(* Logix 5000 project; controller Good_Foods_96985_10252022_1208 vendor 1 type 14 code 151 rev 32.15; software revision 32.04; part 3 of 4 *)
(* tags used below, declared in another part *)
   Active_Container_Recipe : Container_Recipe;
   AG_Index_Sys : BOOL;
   Axis_Virtual_Left_Denest : AXIS_VIRTUAL;
   Axis_Virtual_Right_Denest : AXIS_VIRTUAL;
   bAuto_Axis_Reset : BOOL;
   bAuto_Disable_Servos : BOOL;
   bAuto_Reset_Servos : BOOL;
   bHMI_IND_Servos_Disable : BOOL;
   bHMI_IND_Servos_Enable : BOOL;
   bHMI_PB_Fault_Reset : BOOL;
   bHMI_PB_JogFwd_Left_Denester : BOOL;
   bHMI_PB_JogFwd_Right_Denester : BOOL;
   bHMI_PB_JogRev_Left_Denester : BOOL;
   bHMI_PB_JogRev_Right_Denester : BOOL;
   bHMI_PB_Left_Denester_Enabled : BOOL;
   bHMI_PB_Move_Screws_to_Zero : BOOL;
   bHMI_PB_Park_Denesters : BOOL;
   bHMI_PB_Park_Left_Denester : BOOL;
   bHMI_PB_Park_Right_Denester : BOOL;
   bHMI_PB_Right_Denester_Enabled : BOOL;
   bHMI_PB_Servos_Disable : BOOL;
   bHMI_PB_Servos_Enable : BOOL;
   bHMI_PB_Teach_Zero_Left_Denester : BOOL;
   bHMI_PB_Teach_Zero_Master_Encoder : BOOL;
   bHMI_PB_Teach_Zero_Right_Denester : BOOL;
   bHMI_PB_Zero_All : BOOL;
   bHome_Master_Encoder : BOOL;
   bLeft_Index_Complete : BOOL;
   bLeft_Index_Cycle_Duration : BOOL;
   bLeft_Indexing : BOOL;
   bLeft_System_Not_Running : BOOL;
   bLeftPrimeBacklog_OK : BOOL;
   bMachine_Startup_Delay : BOOL;
   bRight_Index_Complete : BOOL;
   bRight_Index_Cycle_Duration : BOOL;
   bRight_Indexing : BOOL;
   bRight_System_Not_Running : BOOL;
   bRightPrimeBacklog_OK : BOOL;
   bSystem_Active : BOOL;
   bSystem_Alarm_Active : BOOL;
   bSystem_Decouple_CMPLT : BOOL;
   bSystem_Denester_Run_Perm : BOOL;
   bSystem_Gearing_CMPLT : BOOL;
   bSystem_Park_CMPLT : BOOL;
   bSystem_Sync_CMPLT : BOOL;
   CamP_RampDwn : CAM_PROFILE[40];
   CamP_RampUp : CAM_PROFILE[40];
   CamP_Run : CAM_PROFILE[40];
   ctuLeftStartup : COUNTER;
   ctuRightDlyStop : COUNTER;
   DI_Safety_Relay_OK : BOOL;
   dLeft_Denester_Jog_Dir : DINT;
   dRight_Denester_Jog_Dir : DINT;
   dSystem_Start_Seq_CMD : DINT;
   dSystem_Stop_Seq_CMD : DINT;
   dTempRevsTime : DINT;
   Index_Position : INT;
   intLug_Drop_High_Limit : INT;
   Left_Denester : AXIS_CIP_DRIVE;
   Left_Index_Cycle_Duration_Timer : TIMER;
   Left_Index_Measured_Cycle_Time : DINT;
   Left_Not_Running_Timer : TIMER;
   MAFR_Axis_Virtual : MOTION_INSTRUCTION;
   MAFR_Left_Denester : MOTION_INSTRUCTION;
   MAFR_Right_Denester : MOTION_INSTRUCTION;
   MAG_StartGear_LeftDenester : MOTION_INSTRUCTION;
   MAG_StartGear_RightDenester : MOTION_INSTRUCTION;
   MAH_Axis_Virtual : MOTION_INSTRUCTION;
   MAH_Left_Denester : MOTION_INSTRUCTION;
   MAH_Master_Encoder : MOTION_INSTRUCTION;
   MAH_Right_Denester : MOTION_INSTRUCTION;
   MAJ_Left_Denester_Jog : MOTION_INSTRUCTION;
   MAJ_Right_Denester_Jog : MOTION_INSTRUCTION;
   MAM_Home_Left_Denester : MOTION_INSTRUCTION;
   MAM_Home_Right_Denester : MOTION_INSTRUCTION;
   MAM_Left_Denester_Sync : MOTION_INSTRUCTION;
   MAM_Park_Left_Denester : MOTION_INSTRUCTION;
   MAM_Park_Right_Denester : MOTION_INSTRUCTION;
   MAM_Right_Denester_Sync : MOTION_INSTRUCTION;
   mamAxisLeftSCREW_INDEXMOVE : MOTION_INSTRUCTION;
   mamAxisRightSCREW_INDEXMOVE : MOTION_INSTRUCTION;
   MAPC_LeftDenesterToLugBelt_RampDwn : MOTION_INSTRUCTION;
   MAPC_LeftDenesterToLugBelt_RampUp : MOTION_INSTRUCTION;
   MAPC_LeftDenesterToLugBelt_Run : MOTION_INSTRUCTION;
   MAPC_RightDenesterToLugBelt_RampDwn : MOTION_INSTRUCTION;
   MAPC_RightDenesterToLugBelt_RampUp : MOTION_INSTRUCTION;
   MAPC_RightDenesterToLugBelt_Run : MOTION_INSTRUCTION;
   MAS_LeftDenester : MOTION_INSTRUCTION;
   MAS_LeftDenester_Jog : MOTION_INSTRUCTION;
   MAS_LeftDenester_Virtual : MOTION_INSTRUCTION;
   MAS_RightDenester : MOTION_INSTRUCTION;
   MAS_RightDenester_Jog : MOTION_INSTRUCTION;
   MAS_RightDenester_Virtual : MOTION_INSTRUCTION;
   MAS_TEMP_Axis_Master_Follow : MOTION_INSTRUCTION;
   MASR_Axis_Virtual : MOTION_INSTRUCTION;
   MASR_Left_Denester : MOTION_INSTRUCTION;
   MASR_Master_Encoder : MOTION_INSTRUCTION;
   MASR_Right_Denester : MOTION_INSTRUCTION;
   Master_Encoder : AXIS_CIP_DRIVE;
   MRP_Axis_Virtual_Sync_Left : MOTION_INSTRUCTION;
   MRP_Axis_Virtual_Sync_Right : MOTION_INSTRUCTION;
   MSF_Left_Denester : MOTION_INSTRUCTION;
   MSF_Right_Denester : MOTION_INSTRUCTION;
   MSO_Left_Denester : MOTION_INSTRUCTION;
   MSO_Right_Denester : MOTION_INSTRUCTION;
   ONS : DINT[16];
   r_Index_Speed : REAL;
   rHMI_Jog_Speed : REAL;
   Right_Denester : AXIS_CIP_DRIVE;
   Right_Index_Cycle_Duration_Timer : TIMER;
   Right_Index_Measured_Cycle_Time : DINT;
   Right_Not_Running_Timer : TIMER;
   rJog_Speed_Command : DINT;
   rLeft_Actual_Throughput : REAL;
   rLeft_Denester_Actual_Position : REAL;
   rLeft_Denester_Position_High : REAL;
   rLeft_Denester_Position_Low : REAL;
   rMaster_Encoder_Actual_Position : REAL;
   rRight_Actual_Throughput : REAL;
   rRight_Denester_Actual_Position : REAL;
   rRight_Denester_Position_High : DINT;
   rRight_Denester_Position_Low : REAL;
   rSystem_Throughput : REAL;
   rTEMP_Axis_Master_Follow_Actual_Position : REAL;
   rVirtual_Right_Denest_Actual_Position : REAL;
   Screw_Accel : REAL;
   Screw_Decel : REAL;
   Servos : MOTION_GROUP;
   TEMP_Axis_Master_Follow : AXIS_VIRTUAL;
   tMachine_Startup_Delay : TIMER;
   tTempRevs : TIMER;
(* MainProgram, continued *)

ROUTINE _20_Servo_Init   (* ladder *)
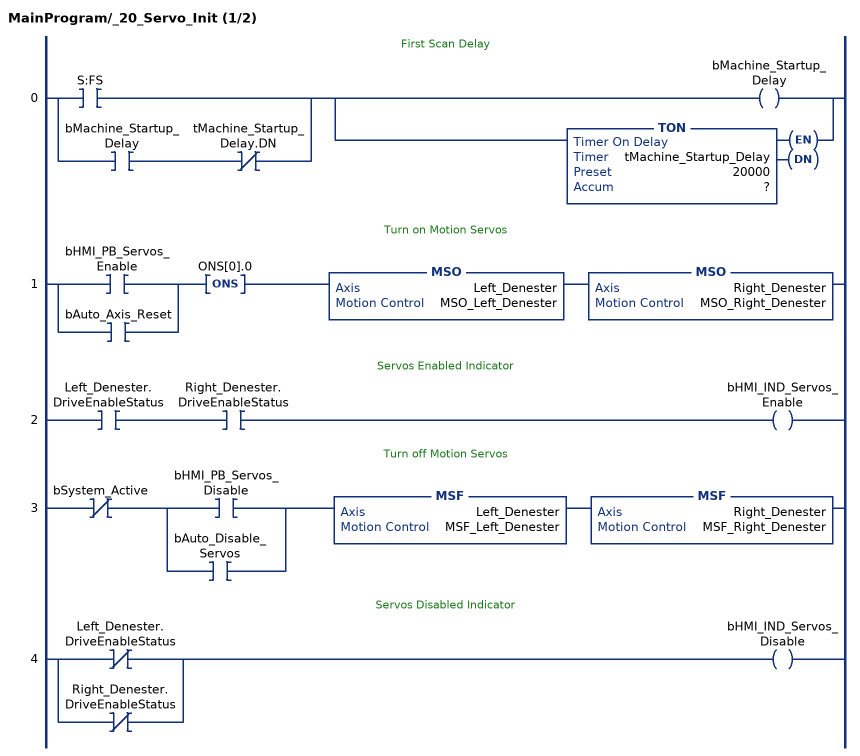
   // First Scan Delay
   0: [XIC(S:FS) ,XIC(bMachine_Startup_Delay) XIO(tMachine_Startup_Delay.DN) ][OTE(bMachine_Startup_Delay) ,TON(tMachine_Startup_Delay,?,?) ];
   // Turn on Motion Servos
   1: [XIC(bHMI_PB_Servos_Enable) ,XIC(bAuto_Axis_Reset) ]ONS(ONS[0].0)MSO(Left_Denester,MSO_Left_Denester)MSO(Right_Denester,MSO_Right_Denester);
   // Servos Enabled Indicator
   2: XIC(Left_Denester.DriveEnableStatus)XIC(Right_Denester.DriveEnableStatus)OTE(bHMI_IND_Servos_Enable);
   // Turn off Motion Servos
   3: XIO(bSystem_Active)[XIC(bHMI_PB_Servos_Disable) ,XIC(bAuto_Disable_Servos) ]MSF(Left_Denester,MSF_Left_Denester)MSF(Right_Denester,MSF_Right_Denester);
   // Servos Disabled Indicator
   4: [XIO(Left_Denester.DriveEnableStatus) ,XIO(Right_Denester.DriveEnableStatus) ]OTE(bHMI_IND_Servos_Disable);
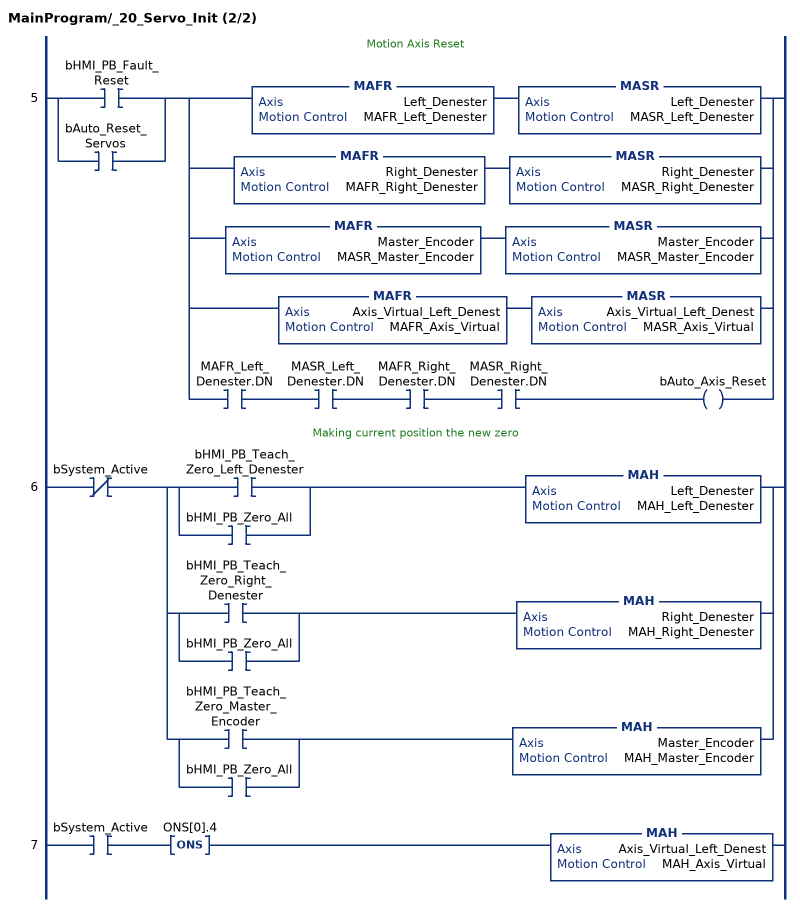
   // Motion Axis Reset
   5: [XIC(bHMI_PB_Fault_Reset) ,XIC(bAuto_Reset_Servos) ][MAFR(Left_Denester,MAFR_Left_Denester) MASR(Left_Denester,MASR_Left_Denester) ,MAFR(Right_Denester,MAFR_Right_Denester) MASR(Right_Denester,MASR_Right_Denester) ,MAFR(Master_Encoder,MASR_Master_Encoder) MASR(Master_Encoder,MASR_Master_Encoder) ,MAFR(Axis_Virtual_Left_Denest,MAFR_Axis_Virtual) MASR(Axis_Virtual_Left_Denest,MASR_Axis_Virtual) ,XIC(MAFR_Left_Denester.DN) XIC(MASR_Left_Denester.DN) XIC(MAFR_Right_Denester.DN) XIC(MASR_Right_Denester.DN) OTE(bAuto_Axis_Reset) ];
   // Making current position the new zero
   6: XIO(bSystem_Active)[[XIC(bHMI_PB_Teach_Zero_Left_Denester) ,XIC(bHMI_PB_Zero_All) ] MAH(Left_Denester,MAH_Left_Denester) ,[XIC(bHMI_PB_Teach_Zero_Right_Denester) ,XIC(bHMI_PB_Zero_All) ] MAH(Right_Denester,MAH_Right_Denester) ,[XIC(bHMI_PB_Teach_Zero_Master_Encoder) ,XIC(bHMI_PB_Zero_All) ] MAH(Master_Encoder,MAH_Master_Encoder) ];
   7: XIC(bSystem_Active)ONS(ONS[0].4)MAH(Axis_Virtual_Left_Denest,MAH_Axis_Virtual);
END_ROUTINE

ROUTINE _25_Servo_Motion   (* ladder *)
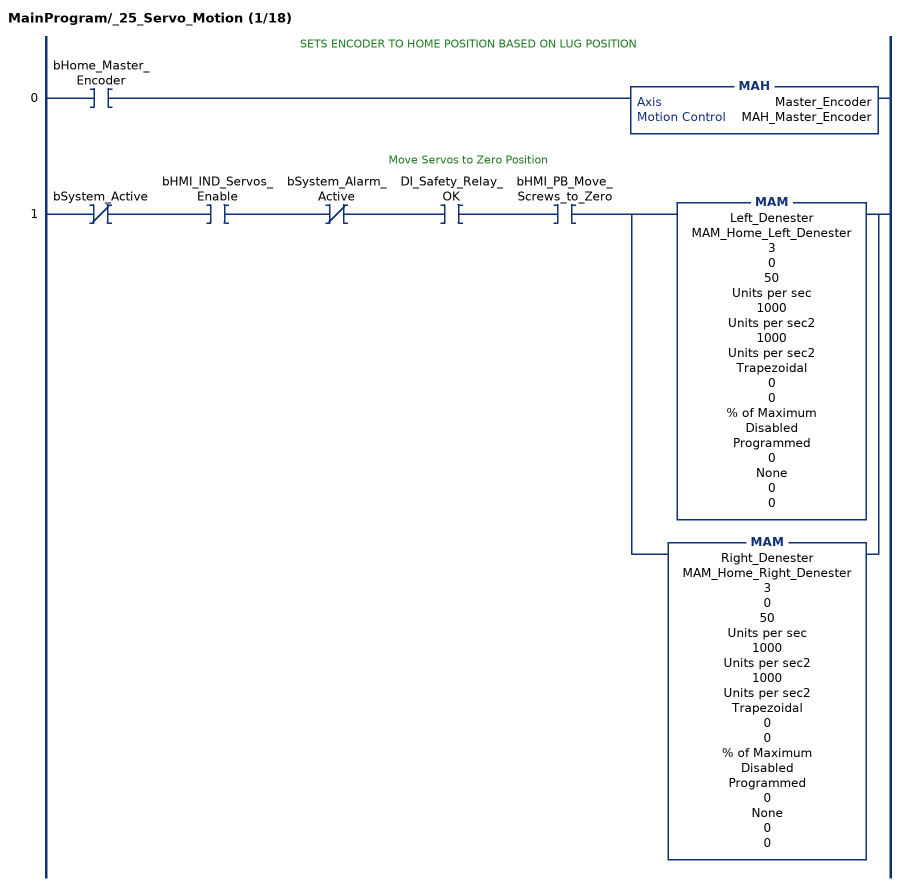
   // SETS ENCODER TO HOME POSITION BASED ON LUG POSITION
   0: XIC(bHome_Master_Encoder)MAH(Master_Encoder,MAH_Master_Encoder);
   // Move Servos to Zero Position
   1: XIO(bSystem_Active)XIC(bHMI_IND_Servos_Enable)XIO(bSystem_Alarm_Active)XIC(DI_Safety_Relay_OK)XIC(bHMI_PB_Move_Screws_to_Zero)[MAM(Left_Denester,MAM_Home_Left_Denester,3,0,50,Units per sec,1000,Units per sec2,1000,Units per sec2,Trapezoidal,0,0,% of Maximum,Disabled,Programmed,0,None,0,0) ,MAM(Right_Denester,MAM_Home_Right_Denester,3,0,50,Units per sec,1000,Units per sec2,1000,Units per sec2,Trapezoidal,0,0,% of Maximum,Disabled,Programmed,0,None,0,0) ];
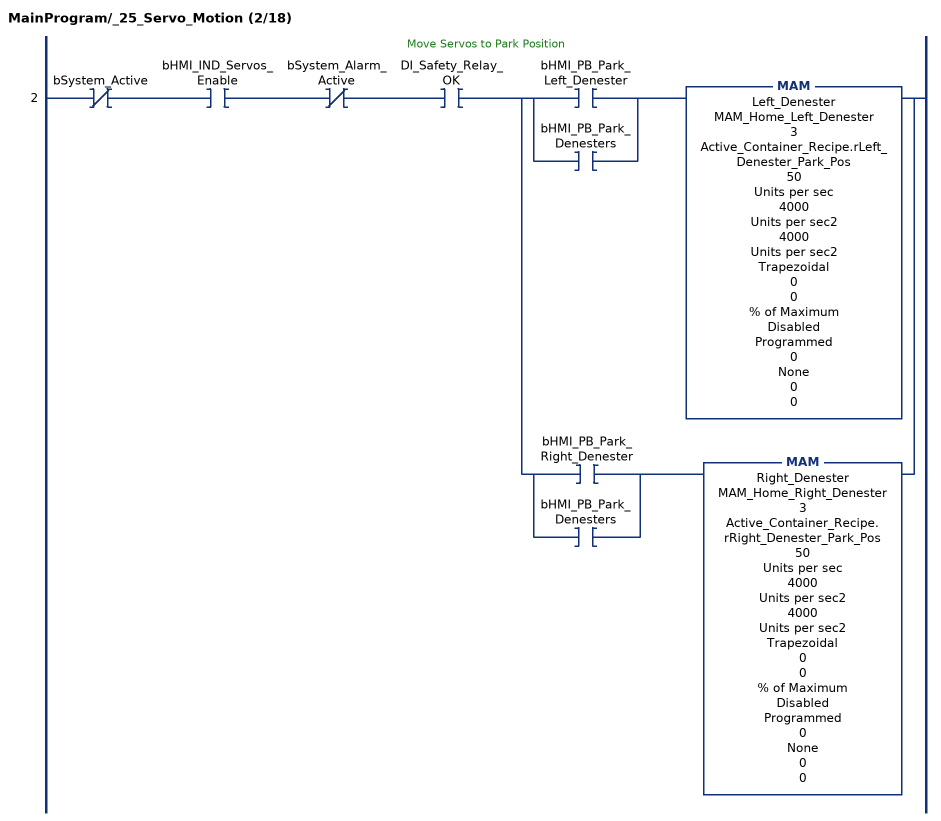
   // Move Servos to Park Position
   2: XIO(bSystem_Active)XIC(bHMI_IND_Servos_Enable)XIO(bSystem_Alarm_Active)XIC(DI_Safety_Relay_OK)[[XIC(bHMI_PB_Park_Left_Denester) ,XIC(bHMI_PB_Park_Denesters) ] MAM(Left_Denester,MAM_Home_Left_Denester,3,Active_Container_Recipe.rLeft_Denester_Park_Pos,50,Units per sec,4000,Units per sec2,4000,Units per sec2,Trapezoidal,0,0,% of Maximum,Disabled,Programmed,0,None,0,0) ,[XIC(bHMI_PB_Park_Right_Denester) ,XIC(bHMI_PB_Park_Denesters) ] MAM(Right_Denester,MAM_Home_Right_Denester,3,Active_Container_Recipe.rRight_Denester_Park_Pos,50,Units per sec,4000,Units per sec2,4000,Units per sec2,Trapezoidal,0,0,% of Maximum,Disabled,Programmed,0,None,0,0) ];
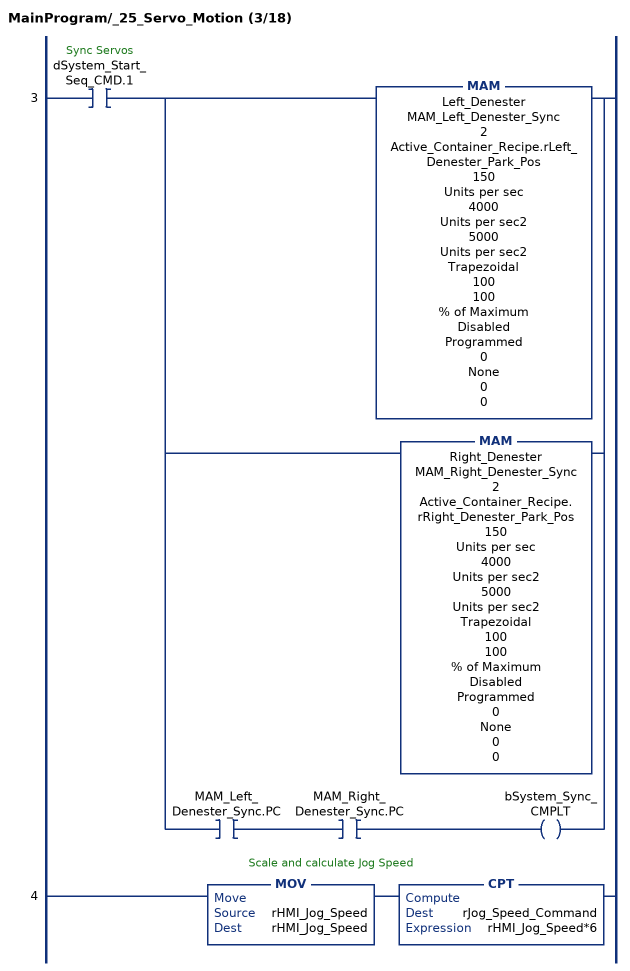
   3: XIC(dSystem_Start_Seq_CMD.1)[MAM(Left_Denester,MAM_Left_Denester_Sync,2,Active_Container_Recipe.rLeft_Denester_Park_Pos,150,Units per sec,4000,Units per sec2,5000,Units per sec2,Trapezoidal,100,100,% of Maximum,Disabled,Programmed,0,None,0,0) ,MAM(Right_Denester,MAM_Right_Denester_Sync,2,Active_Container_Recipe.rRight_Denester_Park_Pos,150,Units per sec,4000,Units per sec2,5000,Units per sec2,Trapezoidal,100,100,% of Maximum,Disabled,Programmed,0,None,0,0) ,XIC(MAM_Left_Denester_Sync.PC) XIC(MAM_Right_Denester_Sync.PC) OTE(bSystem_Sync_CMPLT) ];
   // Scale and calculate Jog Speed
   4: MOV(rHMI_Jog_Speed,rHMI_Jog_Speed)CPT(rJog_Speed_Command,rHMI_Jog_Speed*6);
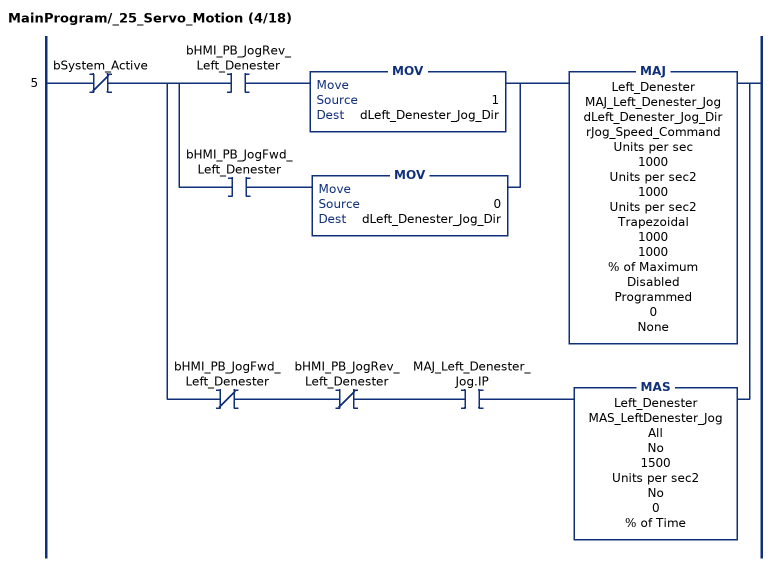
   5: XIO(bSystem_Active)[[XIC(bHMI_PB_JogRev_Left_Denester) MOV(1,dLeft_Denester_Jog_Dir) ,XIC(bHMI_PB_JogFwd_Left_Denester) MOV(0,dLeft_Denester_Jog_Dir) ] MAJ(Left_Denester,MAJ_Left_Denester_Jog,dLeft_Denester_Jog_Dir,rJog_Speed_Command,Units per sec,1000,Units per sec2,1000,Units per sec2,Trapezoidal,1000,1000,% of Maximum,Disabled,Programmed,0,None) ,XIO(bHMI_PB_JogFwd_Left_Denester) XIO(bHMI_PB_JogRev_Left_Denester) XIC(MAJ_Left_Denester_Jog.IP) MAS(Left_Denester,MAS_LeftDenester_Jog,All,No,1500,Units per sec2,No,0,% of Time) ];
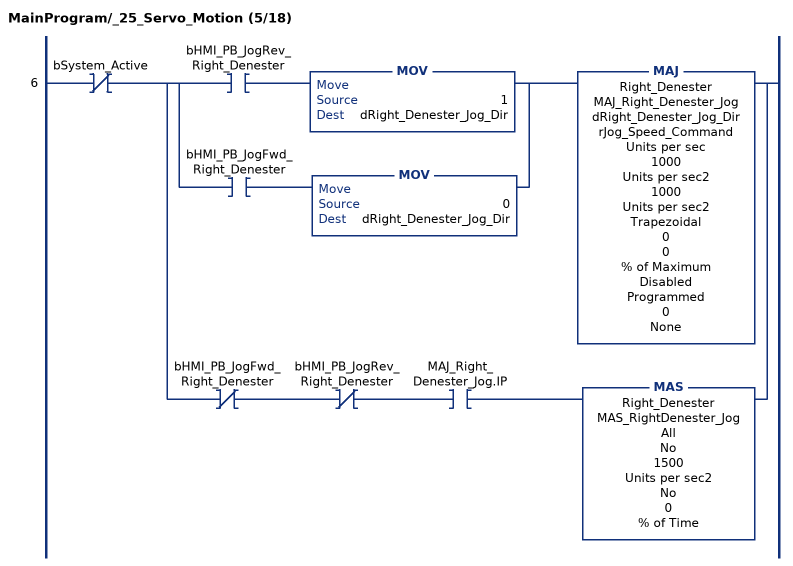
   6: XIO(bSystem_Active)[[XIC(bHMI_PB_JogRev_Right_Denester) MOV(1,dRight_Denester_Jog_Dir) ,XIC(bHMI_PB_JogFwd_Right_Denester) MOV(0,dRight_Denester_Jog_Dir) ] MAJ(Right_Denester,MAJ_Right_Denester_Jog,dRight_Denester_Jog_Dir,rJog_Speed_Command,Units per sec,1000,Units per sec2,1000,Units per sec2,Trapezoidal,0,0,% of Maximum,Disabled,Programmed,0,None) ,XIO(bHMI_PB_JogFwd_Right_Denester) XIO(bHMI_PB_JogRev_Right_Denester) XIC(MAJ_Right_Denester_Jog.IP) MAS(Right_Denester,MAS_RightDenester_Jog,All,No,1500,Units per sec2,No,0,% of Time) ];
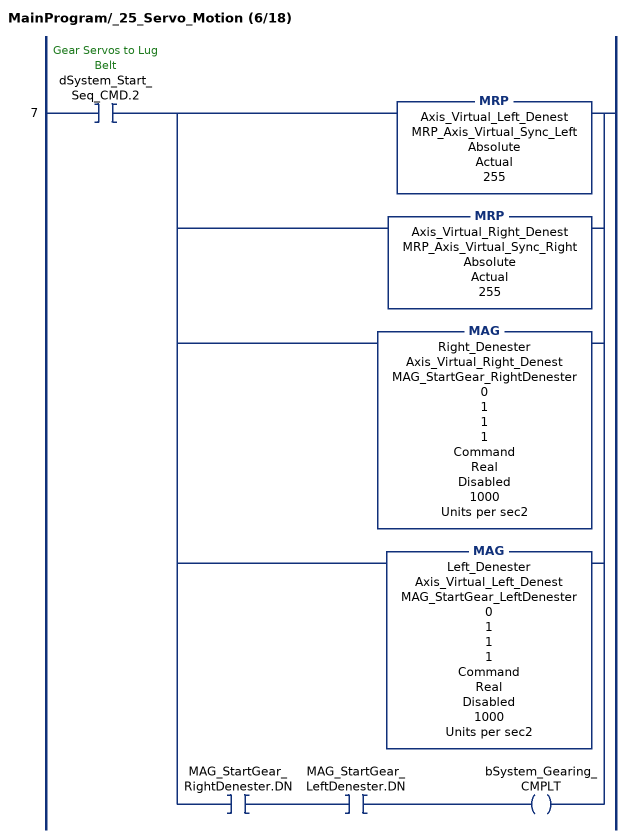
   7: XIC(dSystem_Start_Seq_CMD.2)[MRP(Axis_Virtual_Left_Denest,MRP_Axis_Virtual_Sync_Left,Absolute,Actual,255) ,MRP(Axis_Virtual_Right_Denest,MRP_Axis_Virtual_Sync_Right,Absolute,Actual,255) ,MAG(Right_Denester,Axis_Virtual_Right_Denest,MAG_StartGear_RightDenester,0,1,1,1,Command,Real,Disabled,1000,Units per sec2) ,MAG(Left_Denester,Axis_Virtual_Left_Denest,MAG_StartGear_LeftDenester,0,1,1,1,Command,Real,Disabled,1000,Units per sec2) ,XIC(MAG_StartGear_RightDenester.DN) XIC(MAG_StartGear_LeftDenester.DN) OTE(bSystem_Gearing_CMPLT) ];
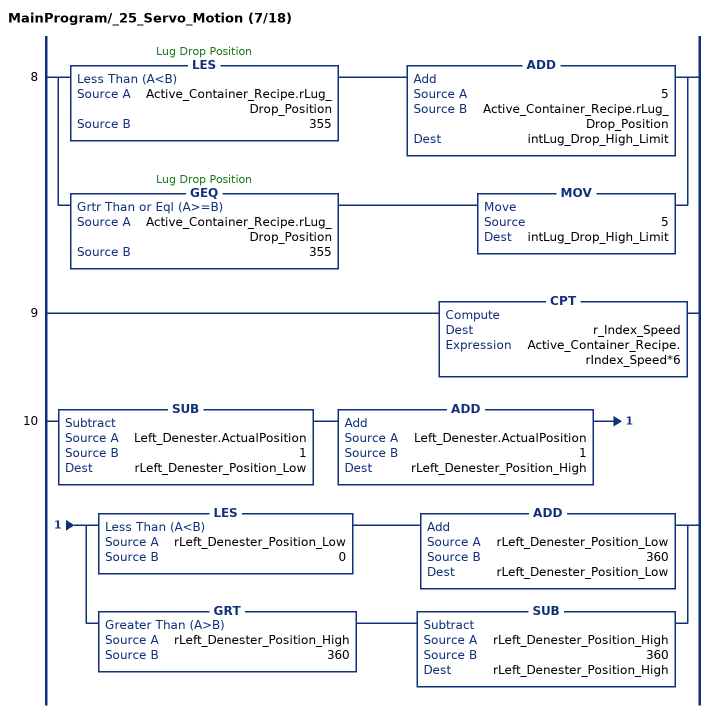
   8: [LES(Active_Container_Recipe.rLug_Drop_Position,355) ADD(5,Active_Container_Recipe.rLug_Drop_Position,intLug_Drop_High_Limit) ,GEQ(Active_Container_Recipe.rLug_Drop_Position,355) MOV(5,intLug_Drop_High_Limit) ];
   9: CPT(r_Index_Speed,Active_Container_Recipe.rIndex_Speed*6);
   10: SUB(Left_Denester.ActualPosition,1,rLeft_Denester_Position_Low)ADD(Left_Denester.ActualPosition,1,rLeft_Denester_Position_High)[LES(rLeft_Denester_Position_Low,0) ADD(rLeft_Denester_Position_Low,360,rLeft_Denester_Position_Low) ,GRT(rLeft_Denester_Position_High,360) SUB(rLeft_Denester_Position_High,360,rLeft_Denester_Position_High) ];
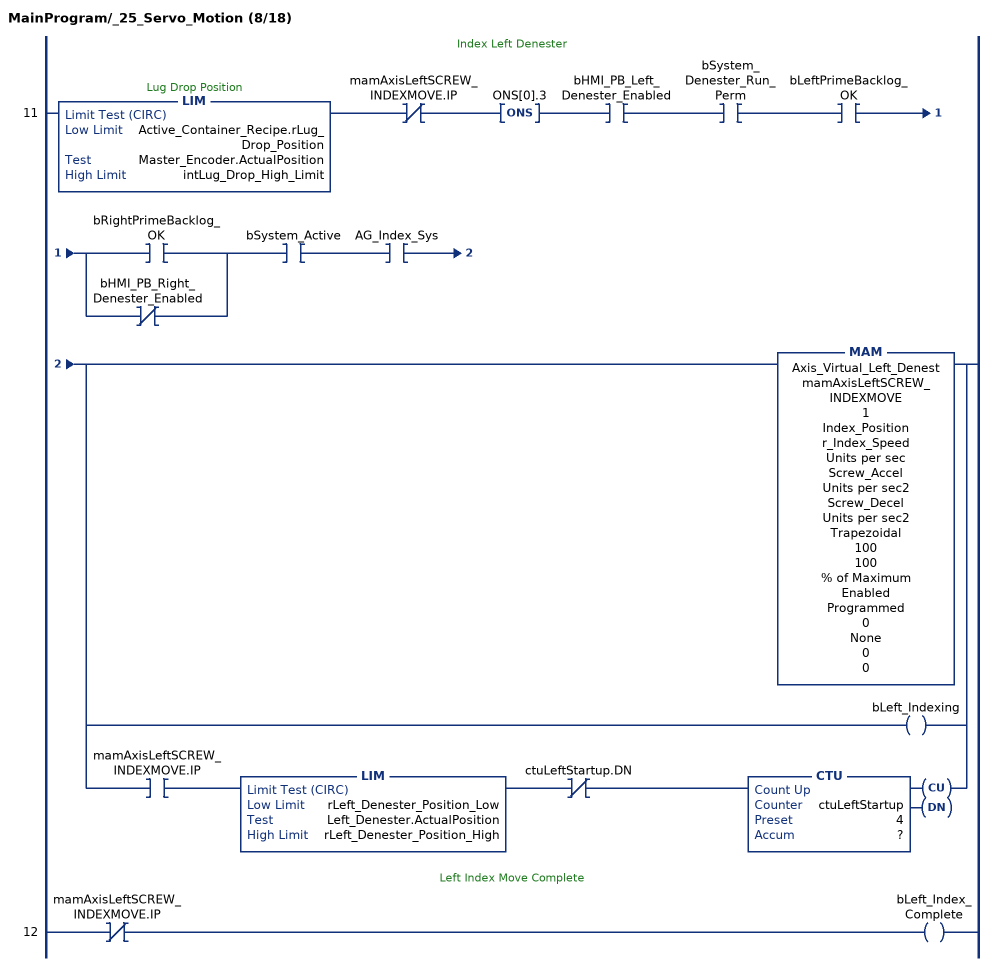
   // Index Left Denester
   11: LIM(Active_Container_Recipe.rLug_Drop_Position,Master_Encoder.ActualPosition,intLug_Drop_High_Limit)XIO(mamAxisLeftSCREW_INDEXMOVE.IP)ONS(ONS[0].3)XIC(bHMI_PB_Left_Denester_Enabled)XIC(bSystem_Denester_Run_Perm)XIC(bLeftPrimeBacklog_OK)[XIC(bRightPrimeBacklog_OK) ,XIO(bHMI_PB_Right_Denester_Enabled) ]XIC(bSystem_Active)XIC(AG_Index_Sys)[MAM(Axis_Virtual_Left_Denest,mamAxisLeftSCREW_INDEXMOVE,1,Index_Position,r_Index_Speed,Units per sec,Screw_Accel,Units per sec2,Screw_Decel,Units per sec2,Trapezoidal,100,100,% of Maximum,Enabled,Programmed,0,None,0,0) ,OTE(bLeft_Indexing) ,XIC(mamAxisLeftSCREW_INDEXMOVE.IP) LIM(rLeft_Denester_Position_Low,Left_Denester.ActualPosition,rLeft_Denester_Position_High) XIO(ctuLeftStartup.DN) CTU(ctuLeftStartup,?,?) ];
   // Left Index Move Complete
   12: XIO(mamAxisLeftSCREW_INDEXMOVE.IP)OTE(bLeft_Index_Complete);
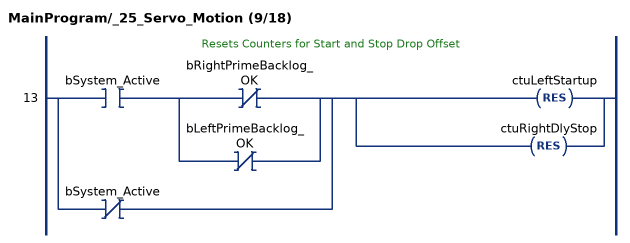
   // Resets Counters for Start and Stop Drop Offset
   13: [XIC(bSystem_Active) [XIO(bRightPrimeBacklog_OK) ,XIO(bLeftPrimeBacklog_OK) ] ,XIO(bSystem_Active) ][RES(ctuLeftStartup) ,RES(ctuRightDlyStop) ];
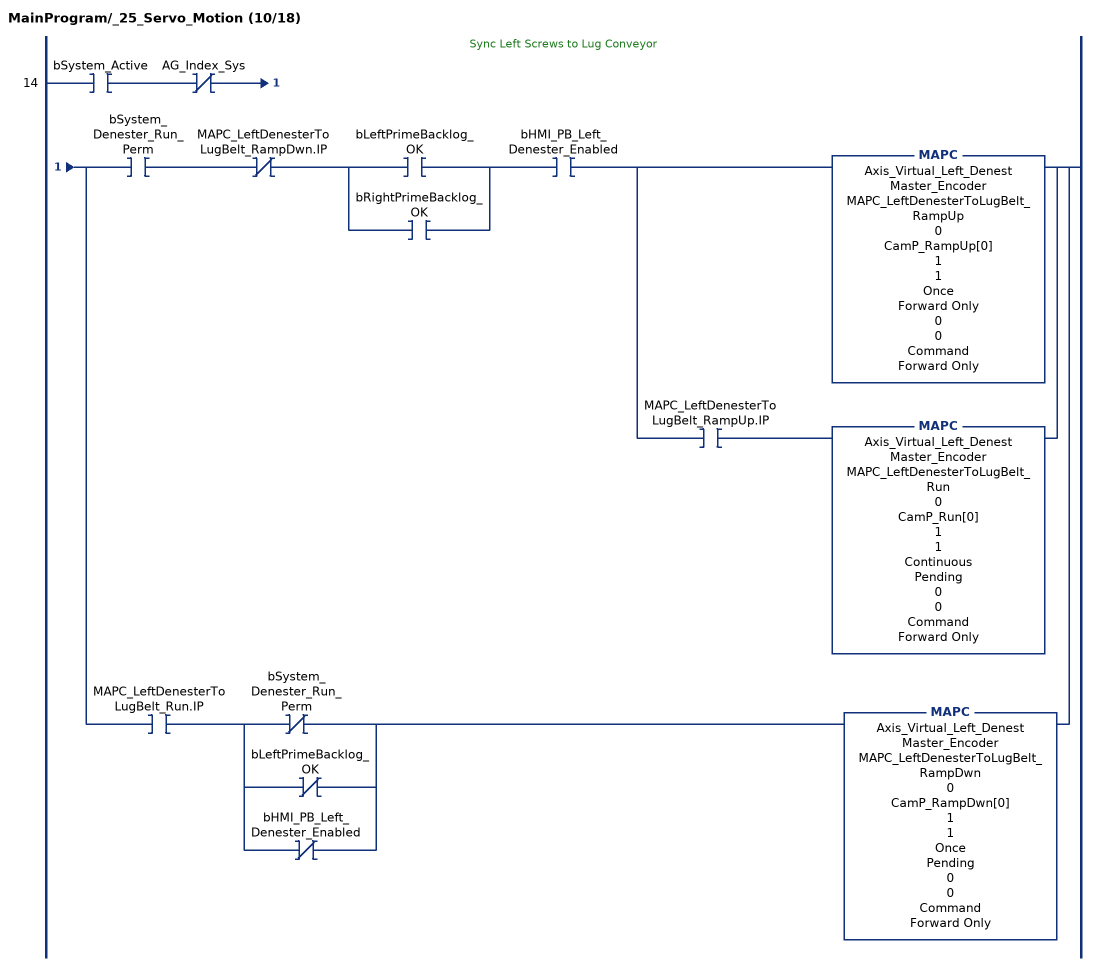
   // Sync Left Screws to Lug Conveyor
   14: XIC(bSystem_Active)XIO(AG_Index_Sys)[XIC(bSystem_Denester_Run_Perm) XIO(MAPC_LeftDenesterToLugBelt_RampDwn.IP) [XIC(bLeftPrimeBacklog_OK) ,XIC(bRightPrimeBacklog_OK) ] XIC(bHMI_PB_Left_Denester_Enabled) [MAPC(Axis_Virtual_Left_Denest,Master_Encoder,MAPC_LeftDenesterToLugBelt_RampUp,0,CamP_RampUp[0],1,1,Once,Forward Only,0,0,Command,Forward Only) ,XIC(MAPC_LeftDenesterToLugBelt_RampUp.IP) MAPC(Axis_Virtual_Left_Denest,Master_Encoder,MAPC_LeftDenesterToLugBelt_Run,0,CamP_Run[0],1,1,Continuous,Pending,0,0,Command,Forward Only) ] ,XIC(MAPC_LeftDenesterToLugBelt_Run.IP) [XIO(bSystem_Denester_Run_Perm) ,XIO(bLeftPrimeBacklog_OK) ,XIO(bHMI_PB_Left_Denester_Enabled) ] MAPC(Axis_Virtual_Left_Denest,Master_Encoder,MAPC_LeftDenesterToLugBelt_RampDwn,0,CamP_RampDwn[0],1,1,Once,Pending,0,0,Command,Forward Only) ];
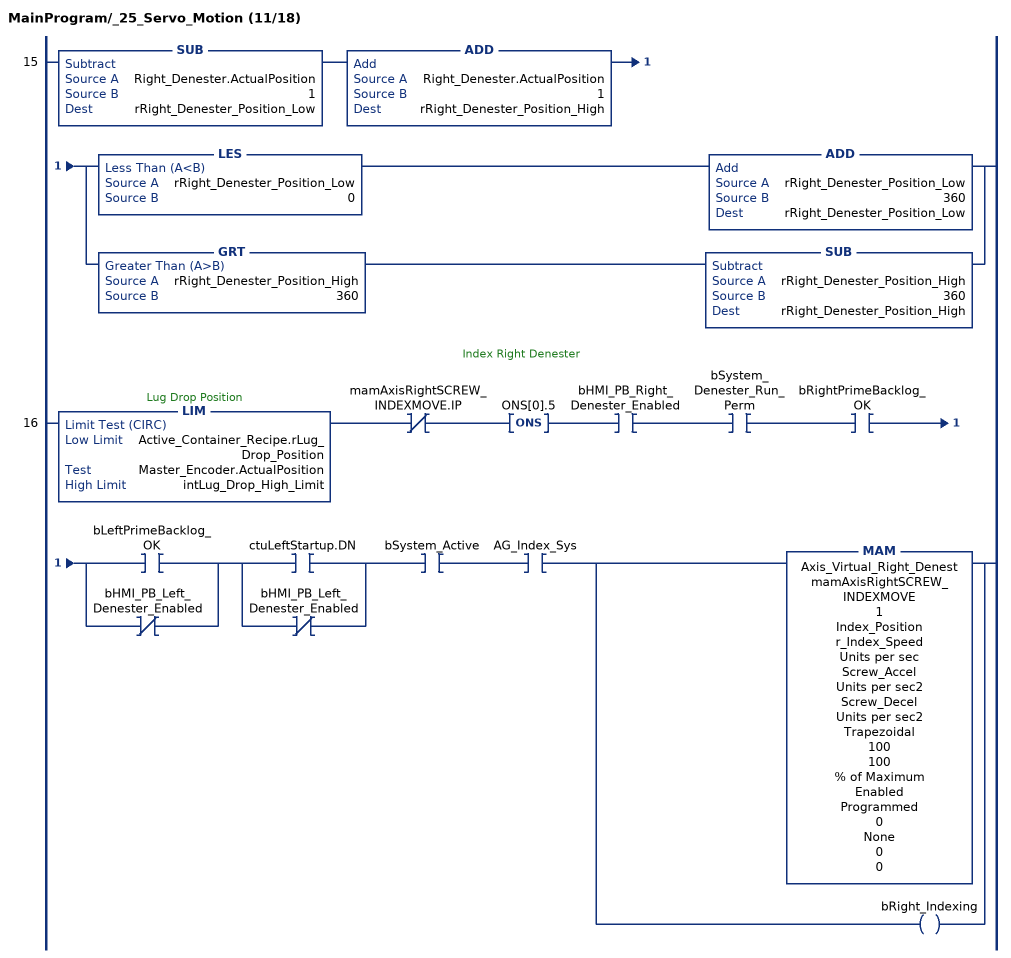
   15: SUB(Right_Denester.ActualPosition,1,rRight_Denester_Position_Low)ADD(Right_Denester.ActualPosition,1,rRight_Denester_Position_High)[LES(rRight_Denester_Position_Low,0) ADD(rRight_Denester_Position_Low,360,rRight_Denester_Position_Low) ,GRT(rRight_Denester_Position_High,360) SUB(rRight_Denester_Position_High,360,rRight_Denester_Position_High) ];
   // Index Right Denester
   16: LIM(Active_Container_Recipe.rLug_Drop_Position,Master_Encoder.ActualPosition,intLug_Drop_High_Limit)XIO(mamAxisRightSCREW_INDEXMOVE.IP)ONS(ONS[0].5)XIC(bHMI_PB_Right_Denester_Enabled)XIC(bSystem_Denester_Run_Perm)XIC(bRightPrimeBacklog_OK)[XIC(bLeftPrimeBacklog_OK) ,XIO(bHMI_PB_Left_Denester_Enabled) ][XIC(ctuLeftStartup.DN) ,XIO(bHMI_PB_Left_Denester_Enabled) ]XIC(bSystem_Active)XIC(AG_Index_Sys)[MAM(Axis_Virtual_Right_Denest,mamAxisRightSCREW_INDEXMOVE,1,Index_Position,r_Index_Speed,Units per sec,Screw_Accel,Units per sec2,Screw_Decel,Units per sec2,Trapezoidal,100,100,% of Maximum,Enabled,Programmed,0,None,0,0) ,OTE(bRight_Indexing) ];
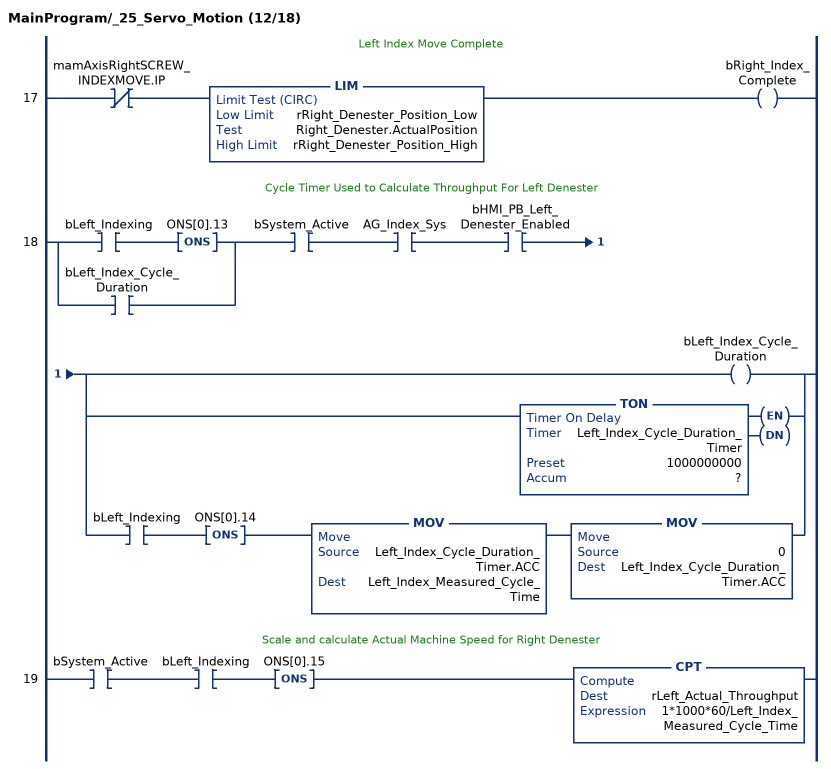
   // Left Index Move Complete
   17: XIO(mamAxisRightSCREW_INDEXMOVE.IP)LIM(rRight_Denester_Position_Low,Right_Denester.ActualPosition,rRight_Denester_Position_High)OTE(bRight_Index_Complete);
   // Cycle Timer Used to Calculate Throughput For Left Denester
   18: [XIC(bLeft_Indexing) ONS(ONS[0].13) ,XIC(bLeft_Index_Cycle_Duration) ]XIC(bSystem_Active)XIC(AG_Index_Sys)XIC(bHMI_PB_Left_Denester_Enabled)[OTE(bLeft_Index_Cycle_Duration) ,TON(Left_Index_Cycle_Duration_Timer,?,?) ,XIC(bLeft_Indexing) ONS(ONS[0].14) MOV(Left_Index_Cycle_Duration_Timer.ACC,Left_Index_Measured_Cycle_Time) MOV(0,Left_Index_Cycle_Duration_Timer.ACC) ];
   // Scale and calculate Actual Machine Speed for Right Denester
   19: XIC(bSystem_Active)XIC(bLeft_Indexing)ONS(ONS[0].15)CPT(rLeft_Actual_Throughput,1*1000*60/Left_Index_Measured_Cycle_Time);
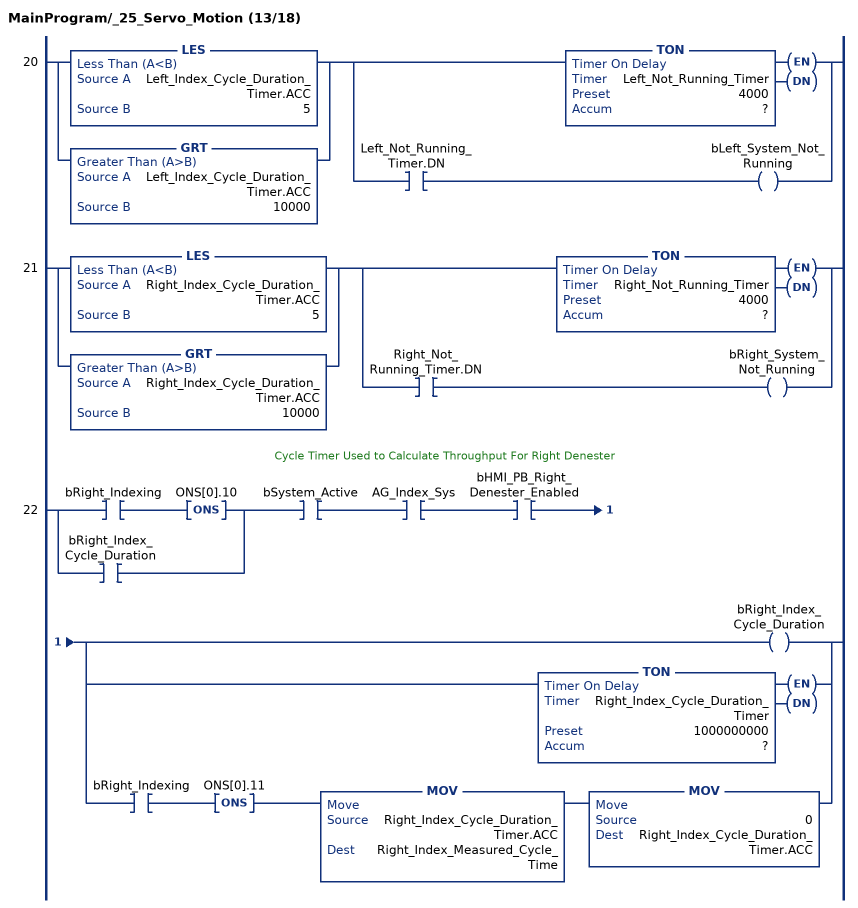
   20: [LES(Left_Index_Cycle_Duration_Timer.ACC,5) ,GRT(Left_Index_Cycle_Duration_Timer.ACC,10000) ][TON(Left_Not_Running_Timer,?,?) ,XIC(Left_Not_Running_Timer.DN) OTE(bLeft_System_Not_Running) ];
   21: [LES(Right_Index_Cycle_Duration_Timer.ACC,5) ,GRT(Right_Index_Cycle_Duration_Timer.ACC,10000) ][TON(Right_Not_Running_Timer,?,?) ,XIC(Right_Not_Running_Timer.DN) OTE(bRight_System_Not_Running) ];
   // Cycle Timer Used to Calculate Throughput For Right Denester
   22: [XIC(bRight_Indexing) ONS(ONS[0].10) ,XIC(bRight_Index_Cycle_Duration) ]XIC(bSystem_Active)XIC(AG_Index_Sys)XIC(bHMI_PB_Right_Denester_Enabled)[OTE(bRight_Index_Cycle_Duration) ,TON(Right_Index_Cycle_Duration_Timer,?,?) ,XIC(bRight_Indexing) ONS(ONS[0].11) MOV(Right_Index_Cycle_Duration_Timer.ACC,Right_Index_Measured_Cycle_Time) MOV(0,Right_Index_Cycle_Duration_Timer.ACC) ];
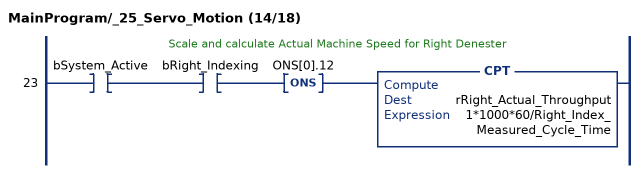
   // Scale and calculate Actual Machine Speed for Right Denester
   23: XIC(bSystem_Active)XIC(bRight_Indexing)ONS(ONS[0].12)CPT(rRight_Actual_Throughput,1*1000*60/Right_Index_Measured_Cycle_Time);
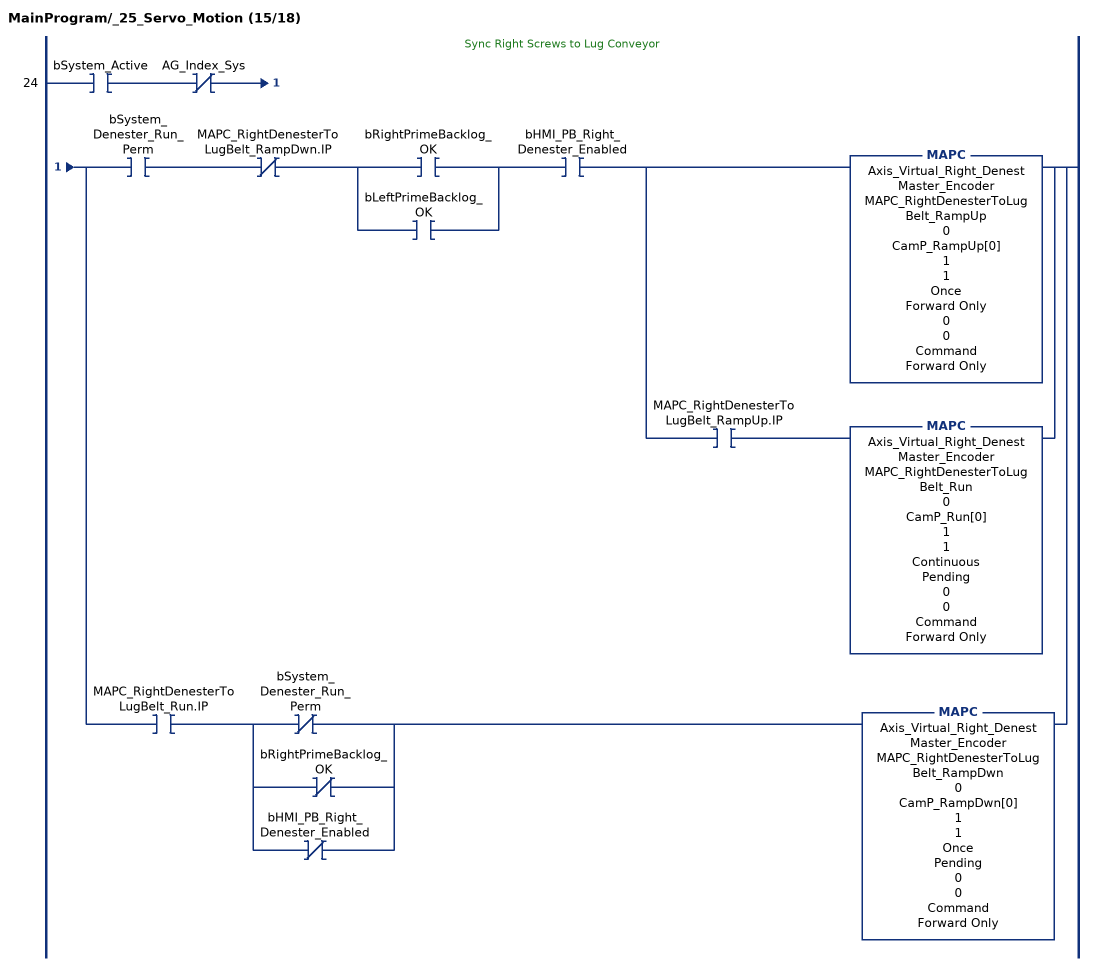
   // Sync Right Screws to Lug Conveyor
   24: XIC(bSystem_Active)XIO(AG_Index_Sys)[XIC(bSystem_Denester_Run_Perm) XIO(MAPC_RightDenesterToLugBelt_RampDwn.IP) [XIC(bRightPrimeBacklog_OK) ,XIC(bLeftPrimeBacklog_OK) ] XIC(bHMI_PB_Right_Denester_Enabled) [MAPC(Axis_Virtual_Right_Denest,Master_Encoder,MAPC_RightDenesterToLugBelt_RampUp,0,CamP_RampUp[0],1,1,Once,Forward Only,0,0,Command,Forward Only) ,XIC(MAPC_RightDenesterToLugBelt_RampUp.IP) MAPC(Axis_Virtual_Right_Denest,Master_Encoder,MAPC_RightDenesterToLugBelt_Run,0,CamP_Run[0],1,1,Continuous,Pending,0,0,Command,Forward Only) ] ,XIC(MAPC_RightDenesterToLugBelt_Run.IP) [XIO(bSystem_Denester_Run_Perm) ,XIO(bRightPrimeBacklog_OK) ,XIO(bHMI_PB_Right_Denester_Enabled) ] MAPC(Axis_Virtual_Right_Denest,Master_Encoder,MAPC_RightDenesterToLugBelt_RampDwn,0,CamP_RampDwn[0],1,1,Once,Pending,0,0,Command,Forward Only) ];
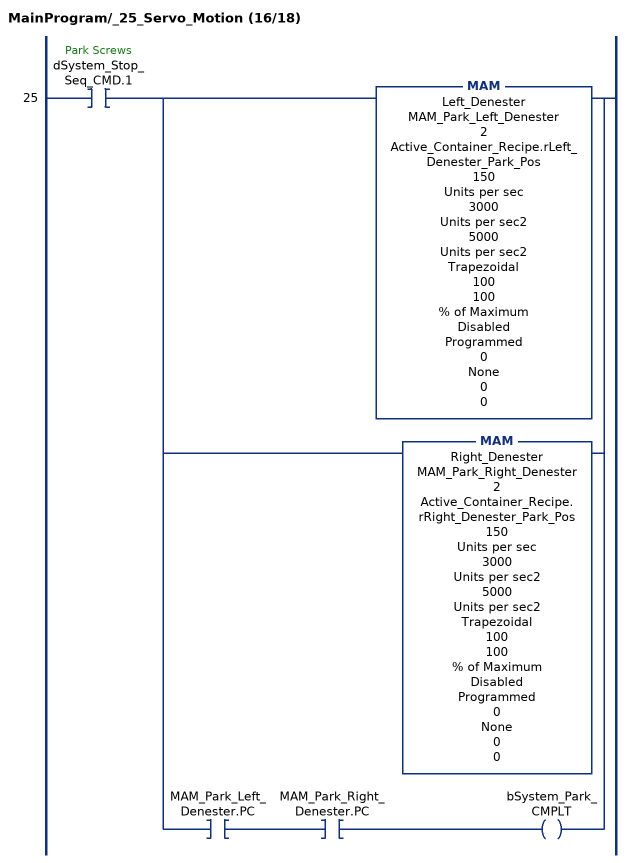
   25: XIC(dSystem_Stop_Seq_CMD.1)[MAM(Left_Denester,MAM_Park_Left_Denester,2,Active_Container_Recipe.rLeft_Denester_Park_Pos,150,Units per sec,3000,Units per sec2,5000,Units per sec2,Trapezoidal,100,100,% of Maximum,Disabled,Programmed,0,None,0,0) ,MAM(Right_Denester,MAM_Park_Right_Denester,2,Active_Container_Recipe.rRight_Denester_Park_Pos,150,Units per sec,3000,Units per sec2,5000,Units per sec2,Trapezoidal,100,100,% of Maximum,Disabled,Programmed,0,None,0,0) ,XIC(MAM_Park_Left_Denester.PC) XIC(MAM_Park_Right_Denester.PC) OTE(bSystem_Park_CMPLT) ];
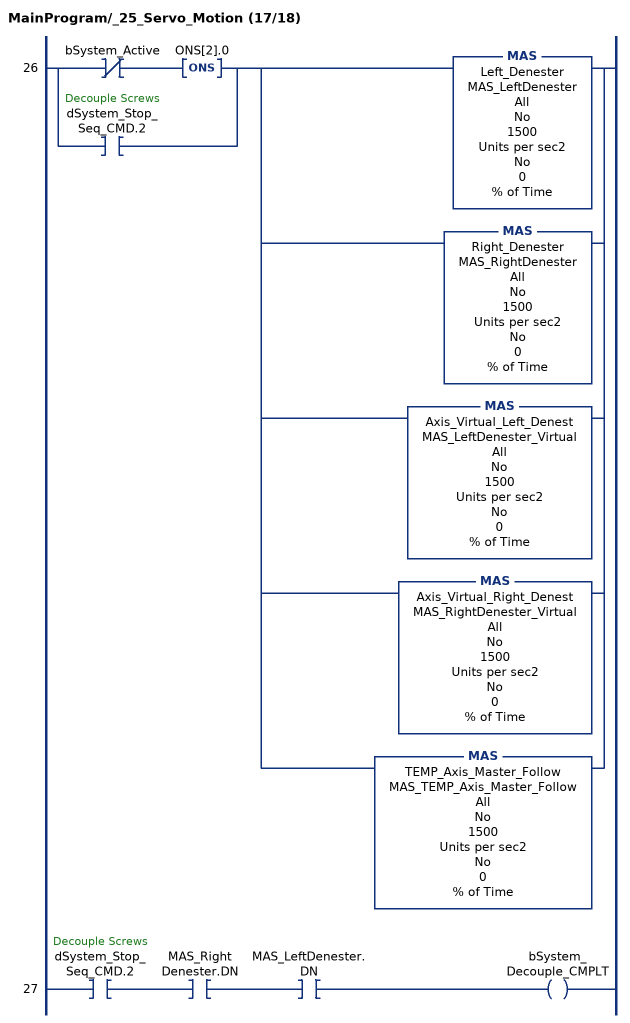
   26: [XIO(bSystem_Active) ONS(ONS[2].0) ,XIC(dSystem_Stop_Seq_CMD.2) ][MAS(Left_Denester,MAS_LeftDenester,All,No,1500,Units per sec2,No,0,% of Time) ,MAS(Right_Denester,MAS_RightDenester,All,No,1500,Units per sec2,No,0,% of Time) ,MAS(Axis_Virtual_Left_Denest,MAS_LeftDenester_Virtual,All,No,1500,Units per sec2,No,0,% of Time) ,MAS(Axis_Virtual_Right_Denest,MAS_RightDenester_Virtual,All,No,1500,Units per sec2,No,0,% of Time) ,MAS(TEMP_Axis_Master_Follow,MAS_TEMP_Axis_Master_Follow,All,No,1500,Units per sec2,No,0,% of Time) ];
   27: XIC(dSystem_Stop_Seq_CMD.2)XIC(MAS_RightDenester.DN)XIC(MAS_LeftDenester.DN)OTE(bSystem_Decouple_CMPLT);
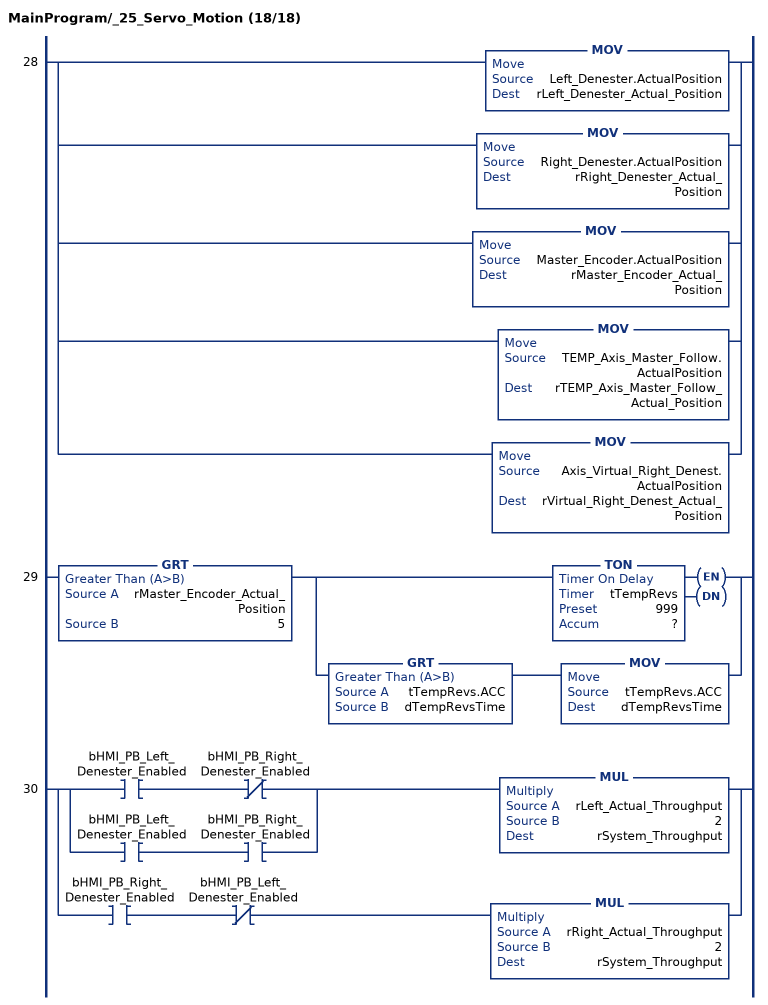
   28: [MOV(Left_Denester.ActualPosition,rLeft_Denester_Actual_Position) ,MOV(Right_Denester.ActualPosition,rRight_Denester_Actual_Position) ,MOV(Master_Encoder.ActualPosition,rMaster_Encoder_Actual_Position) ,MOV(TEMP_Axis_Master_Follow.ActualPosition,rTEMP_Axis_Master_Follow_Actual_Position) ,MOV(Axis_Virtual_Right_Denest.ActualPosition,rVirtual_Right_Denest_Actual_Position) ];
   29: GRT(rMaster_Encoder_Actual_Position,5)[TON(tTempRevs,?,?) ,GRT(tTempRevs.ACC,dTempRevsTime) MOV(tTempRevs.ACC,dTempRevsTime) ];
   30: [[XIC(bHMI_PB_Left_Denester_Enabled) XIO(bHMI_PB_Right_Denester_Enabled) ,XIC(bHMI_PB_Left_Denester_Enabled) XIC(bHMI_PB_Right_Denester_Enabled) ] MUL(rLeft_Actual_Throughput,2,rSystem_Throughput) ,XIC(bHMI_PB_Right_Denester_Enabled) XIO(bHMI_PB_Left_Denester_Enabled) MUL(rRight_Actual_Throughput,2,rSystem_Throughput) ];
END_ROUTINE
